// TIA Portal V17 export
// export: Created 2025-06-26T06:49:15.4222938Z, ExportSetting WithDefaults, DisplayName Totally Integrated Automation Portal, DisplayVersion V17 Update 8, DisplayName TIA Portal Openness, DisplayVersion V17 Update 8, DisplayName TIA Portal Version Control Interface, DisplayVersion V17, DisplayName STEP 7 Professional, DisplayVersion V17 Update 8, DisplayName STEP 7 Safety, DisplayVersion V17 Update 6, DisplayName WinCC Advanced, DisplayVersion V17 Update 8
FUNCTION_BLOCK "fbPWMController"   // FB35, FBD
TITLE = PWM Controller
{ S7_Optimized_Access := 'TRUE' }
VERSION : 0.1
// stored: AutoNumber true, IsIECCheckEnabled false, IsRetainMemResEnabled false, MemoryReserve 0, SetENOAutomatically false, UDAEnableTagReadback false
   VAR_INPUT
      bEnable : Bool;   // 1 = enable controller, 0 = disable
      tOnTime : Time;
      tPeriod : Time;
   END_VAR
   VAR_OUTPUT
      bOut : Bool;
      tOnTimeElapsed : Time;
      tPeriodElapsed : Time;
   END_VAR
   VAR
      PeriodTimer { S7_SetPoint := 'True'} : TP_TIME;
      OnTimer : TP_TIME;
      bOnTime { S7_SetPoint := 'True'} : Bool := True;
   END_VAR
BEGIN

REGION Network 1: Trigger the output
   // Note: if output should start LOW, set initial value of bOnTime to FALSE
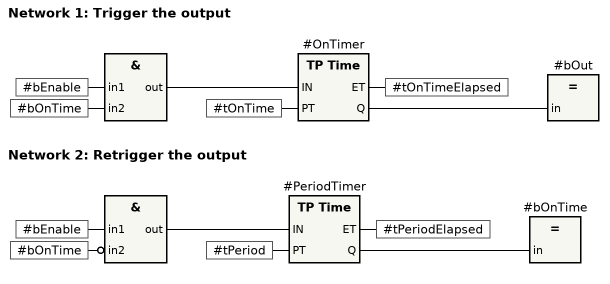
   #OnTimer(IN := #bEnable AND #bOnTime, PT := #tOnTime, ET => #tOnTimeElapsed);   // TP
   #bOut := #OnTimer.Q;
END_REGION

REGION Network 2: Retrigger the output
   #PeriodTimer(IN := #bEnable AND NOT #bOnTime, PT := #tPeriod, ET => #tPeriodElapsed);   // TP
   #bOnTime := #PeriodTimer.Q;
END_REGION

REGION Network 3 (SCL): Reset
   IF #bEnable = FALSE THEN
       RESET_TIMER(#PeriodTimer);
       RESET_TIMER(#OnTimer);
   END_IF;
END_REGION
END_FUNCTION_BLOCK
